FUNCTION_BLOCK ValveBase (* Composite Function Block Type *)
  (* Standard: 61499-2 *)
  (* Version 1.0.1, 10/17/2023, ApplicationLibDevTeam, Schneider Electric, First Version *)
  PACKAGE Main;
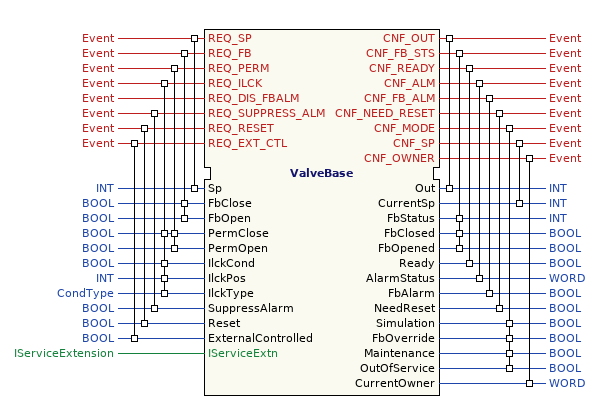
  EVENT_INPUT
    REQ_SP WITH Sp; (* Request to update setpoint *)
    REQ_FB WITH FbClose, FbOpen; (* Request to update feedbacks *)
    REQ_PERM WITH PermClose, PermOpen; (* Request to update permissive conditions *)
    REQ_ILCK WITH PermClose, IlckCond, IlckPos, IlckType; (* Request to update interlock conditions *)
    REQ_DIS_FBALM; (* Request to disable feedback alarm *)
    REQ_SUPPRESS_ALM WITH SuppressAlarm; (* Request to update the alarm suppress status *)
    REQ_RESET WITH Reset; (* Request to reset the device *)
    REQ_EXT_CTL WITH ExternalControlled;
  END_EVENT
  EVENT_OUTPUT
    CNF_OUT WITH Out; (* Execution of confirmation output *)
    CNF_FB_STS WITH FbStatus, FbOpened, FbClosed; (* Execution of confirmed state *)
    CNF_READY WITH Ready; (* Execution of Ready status *)
    CNF_ALM WITH AlarmStatus; (* Execution of confirmation  alarm conditions *)
    CNF_FB_ALM WITH FbAlarm; (* Execution of confirmation  Fb alarm *)
    CNF_NEED_RESET WITH NeedReset; (* Request for Reset *)
    CNF_MODE WITH OutOfService, Simulation, FbOverride, Maintenance; (* Excecution of new operational modes *)
    CNF_SP WITH CurrentSp;
    CNF_OWNER WITH CurrentOwner; (* Execution confirmation of owner *)
  END_EVENT
  VAR_INPUT
    Sp : INT; (* Setpoint of device (1 = Open, 2 = Close) *)
    FbClose : BOOL; (* 1 = Device Close feedback active *)
    FbOpen : BOOL; (* 1 = Device Open feedback active *)
    PermClose : BOOL := TRUE; (* 1 = Device Close permission active *)
    PermOpen : BOOL := TRUE; (* 1 = Device Open permission active *)
    IlckCond : BOOL; (* 1 = Interlock condition active *)
    IlckPos : INT; (* Interlock setpoint state (0 = stop, 1 = Open, 2 = Close, 3 = Interlock inactive) *)
    IlckType : CondType; (* Type of condition interlock, (0 = Normal, 1 = Process interlock/Sequence interlock) *)
    SuppressAlarm : BOOL; (* 1 = Suppress alarm in HMI *)
    Reset : BOOL; (* 1 = Reset device failure *)
    ExternalControlled : BOOL; (* 1 = External control is active *)
  END_VAR
  VAR_OUTPUT
    Out : INT; (* Output to HW ( 1 = Open command, 2 = Close command) depending on NO/NC *)
    CurrentSp : INT; (* Output value considering permissive conditions *)
    FbStatus : INT; (* Confirmed state of the device (0 = Stopped, 1 = Opened, 2 = Closed , 253 = Unknown) *)
    FbClosed : BOOL; (* 1 = Closed *)
    FbOpened : BOOL; (* 1 = Opened *)
    Ready : BOOL; (* 1 = Device is ready to run *)
    AlarmStatus : WORD; (* Bit 2 = Feedback failure status *)
    FbAlarm : BOOL; (* 1 = Feedback failure alarm is active *)
    NeedReset : BOOL; (* 1 = Device need reset to resume the operation *)
    Simulation : BOOL; (* 1 = Simulation mode is active *)
    FbOverride : BOOL; (* 1 = Feedback overide (Sp = FbStatus) *)
    Maintenance : BOOL; (* 1 = Maintenance mode is active *)
    OutOfService : BOOL; (* 1 = Out of service mode is active *)
    CurrentOwner : WORD; (* Current owner data from externlal source and basic owner 16#8 = Program owner, 16#10 = Operator owner, 16#4 = program Local and 16#40 Operator Local *)
  END_VAR
  SOCKETS
    IServiceExtn : IServiceExtension(ServiceState := TRUE); (* Services extension adapter(Seq control, Local panel, Maintenance and Owner) *)
  END_SOCKETS
  (* Alarm Managment *)
  (* Data exchange with sequence *)
  (* Initialization *)
  (* Supervision Interface *)
  (* Owner & Setpoint Management *)
  (* Control *)
  FBS
    plcStart : plcStart(Delay := T#0ms, Prio := 16); {SET_ATTRIBUTE(Configuration.Component.HideUnusedPorts, )}
    spSelection : devInSel(EnBumpless1 := FALSE, EnBumpless2 := TRUE, EnBumpless3 := TRUE, ResetSp := (value:=0,quality:=16#0,timestamp:=LDT#2023-01-20-10:13:38,picosecs:=0), InitialVal := (value:=1,quality:=16#0,timestamp:=LDT#2023-08-11-12:54:59,picosecs:=0)); {SET_ATTRIBUTE(Configuration.Component.HideUnusedPorts, )}
    control : valveLogic;
    feedbackFailure : stateAlarmBasic(AlarmState := TRUE); {SET_ATTRIBUTE(Configuration.Component.HideUnusedPorts, )} {SET_ATTRIBUTE(HMI.AlarmText, $key:SE.App2CommonProcess.AlmLableFbFail)}
    progSpSelection : SELECT_24363B89CFDE21263; {SET_ATTRIBUTE(Configuration.GenericFBType.InterfaceParams, Runtime.Standard#CNT:=2;SELECT:BOOL;IN${CNT$}:INT)}
    IThis : ValveBase_HMI(QI := TRUE);
    basicOwner : ownerControl;
    resetConditions : DS_SELECTX_1579ED5B8ACDFC94C; {SET_ATTRIBUTE(Configuration.GenericFBType.InterfaceParams, Runtime.Standard#CNTX:=3;CNTY:=1;DI${CNTX,_,CNTY$}:BOOL)}
  END_FBS
  EVENT_CONNECTIONS
    control.CNF_FB_ALM TO CNF_FB_ALM;
    control.CNF_FB_STS TO CNF_FB_STS;
    control.CNF_MODE TO CNF_MODE;
    REQ_FB TO control.REQ_FB;
    REQ_DIS_FBALM TO control.REQ_PARA;
    REQ_PERM TO spSelection.REQ_SEL;
    basicOwner.CNF_OWNER TO spSelection.REQ_SEL;
    control.CNF_NEED_RESET TO CNF_NEED_RESET;
    control.CNF_READY TO CNF_READY;
    control.CNF_FB_ALM TO feedbackFailure.REQ;
    control.CNF_ALM TO CNF_ALM;
    control.CNF_OUT TO IServiceExtn.CNF_STATUS;
    control.CNF_FB_STS TO IServiceExtn.CNF_STATUS;
    control.CNF_READY TO IServiceExtn.CNF_READY;
    control.CNF_MODE TO IServiceExtn.CNF_OPMODE;
    REQ_SUPPRESS_ALM TO IServiceExtn.CNF_SUPPRESS_ALM;
    feedbackFailure.INITO TO plcStart.ACK_FIRST;
    plcStart.FIRST_INIT TO IServiceExtn.CNF_SERVICE;
    control.CNF_ILCK TO spSelection.REQ_SEL;
    REQ_SUPPRESS_ALM TO feedbackFailure.REQ_SUPRESS;
    control.CNF_OUT TO CNF_OUT;
    REQ_ILCK TO control.REQ_ILCK;
    spSelection.CNF TO control.REQ_SP;
    IServiceExtn.REQ_OWNER TO basicOwner.REQ_STDOWNER;
    REQ_PERM TO IServiceExtn.CNF_READY;
    control.CNF_DEFAULT_STATE TO spSelection.REQ_SP1;
    REQ_SP TO progSpSelection.REQ;
    IServiceExtn.REQ_CMD TO progSpSelection.REQ;
    progSpSelection.CNF TO spSelection.REQ_SP3;
    control.CNF_ILCK TO IServiceExtn.CNF_READY;
    control.CNF_SP TO CNF_SP;
    control.CNF_ALM TO IServiceExtn.CNF_READY;
    REQ_EXT_CTL TO control.REQ_EXT_CTL;
    basicOwner.CNF_OWNER TO CNF_OWNER;
    REQ_RESET TO resetConditions.REQ3;
    IServiceExtn.REQ_RESET TO resetConditions.REQ2;
    resetConditions.IND TO control.REQ_RESET;
    control.CNF_NEED_RESET TO IServiceExtn.CNF_READY;
    control.CNF_DEFAULT_STATE TO IServiceExtn.CNF_DEFAULT_STATE;
    plcStart.FIRST_INIT TO IThis.34A017503AC1070A;
    IThis.377462E9CE5193B5 TO IThis.F2953B6BB9388F21;
    control.CNF_OUT TO IThis.EC791CA6E67D66B3;
    control.CNF_FB_STS TO IThis.EC791CA6E67D66B3;
    control.CNF_NEED_RESET TO IThis.EC791CA6E67D66B3;
    spSelection.CNF TO IThis.EC791CA6E67D66B3;
    control.CNF_TRANS_FB TO IThis.EC791CA6E67D66B3;
    REQ_SUPPRESS_ALM TO IThis.EC791CA6E67D66B3;
    feedbackFailure.CNF_ALM TO IThis.EC791CA6E67D66B3;
    control.CNF_ILCK TO IThis.EC791CA6E67D66B3;
    REQ_PERM TO IThis.EC791CA6E67D66B3;
    basicOwner.CNF_OWNER TO IThis.EC791CA6E67D66B3;
    control.CNF_SP TO IThis.EC791CA6E67D66B3;
    REQ_EXT_CTL TO IThis.EC791CA6E67D66B3;
    IThis.377462E9CE5193B5 TO feedbackFailure.INIT;
    IThis.377462E9CE5193B5 TO basicOwner.REQ_BASICOWNER;
    IThis.95BEA68906019444 TO feedbackFailure.REQ_PARA;
    IThis.95BEA68906019444 TO control.REQ_DEFAULT_STATE;
    IThis.95BEA68906019444 TO control.REQ_PARA;
    IThis.95BEA68906019444 TO IServiceExtn.CNF_CFG;
    IThis.C6CA4032A5F6989A TO spSelection.REQ_SP2;
    IThis.1A2B085F4B246BF1 TO resetConditions.REQ1;
    IThis.4711DA9A2DFC024 TO control.REQ_PARA;
    IThis.4711DA9A2DFC024 TO spSelection.REQ_SEL;
    IThis.4711DA9A2DFC024 TO basicOwner.REQ_FORCE;
    IThis.AB45C9C76752120B TO basicOwner.REQ_BASICOWNER;
    control.CNF_SP TO IServiceExtn.CNF_STATUS;
  END_CONNECTIONS
  DATA_CONNECTIONS
    control.FbAlarm TO FbAlarm;
    control.Mode TO IServiceExtn.OpMode;
    SuppressAlarm TO feedbackFailure.Suppress;
    control.FbAlarm TO feedbackFailure.Input;
    IlckType TO control.IlckType;
    FbClose TO control.FbClose;
    FbOpen TO control.FbOpen;
    control.FbClosed TO FbClosed;
    control.FbOpened TO FbOpened;
    control.FbStatus TO FbStatus;
    control.NeedReset TO NeedReset;
    control.Ready TO Ready;
    control.Alarm TO AlarmStatus;
    control.CurrentSp TO CurrentSp;
    control.FbStatus TO IServiceExtn.Status;
    control.CurrentSp TO IServiceExtn.CurrentSp;
    control.CurrentOut TO IServiceExtn.CurrentOp;
    control.NeedReset TO IServiceExtn.NeedReset;
    control.Ready TO IServiceExtn.Ready;
    SuppressAlarm TO IServiceExtn.SuppressAlarm;
    control.CondPos TO spSelection.IlckSp;
    control.Interlocked TO spSelection.Ilck;
    control.Out TO Out;
    IlckPos TO control.IlckPos;
    PermClose TO spSelection.PermActive2;
    IlckCond TO control.IlckCond;
    IServiceExtn.StdOwner TO basicOwner.StdOwner;
    basicOwner.OperatorOwner TO spSelection.Sel2;
    basicOwner.ProgramOwner TO spSelection.Sel3;
    control.Alarm TO IServiceExtn.Alarm;
    control.Interlocked TO IServiceExtn.Interlocked;
    PermOpen TO IServiceExtn.PermActive1;
    PermClose TO IServiceExtn.PermActive2;
    PermClose TO spSelection.PermPassive;
    control.DefaultState TO spSelection.Val1;
    basicOwner.StdOwnerConnected TO progSpSelection.SELECT;
    Sp TO progSpSelection.IN1;
    IServiceExtn.Sp TO progSpSelection.IN2;
    progSpSelection.OUT TO spSelection.Val3;
    spSelection.PermVal TO control.Sp;
    PermClose TO IServiceExtn.PermPassive;
    ExternalControlled TO control.ExternalControlled;
    basicOwner.Owner TO CurrentOwner;
    Reset TO resetConditions.DI3_1;
    IServiceExtn.Reset TO resetConditions.DI2_1;
    resetConditions.OUT1 TO control.Reset;
    control.DefaultState TO IServiceExtn.DefaultState;
    PermOpen TO spSelection.PermActive1;
    control.FbStatus TO IThis.F2AD3CD6DCE76874;
    control.TransFbStatus TO IThis.18339E8B84CEF55;
    control.CurrentOut TO IThis.D2C35BC47DF71FCC;
    control.CurrentSp TO IThis.C6876D790F3A950E;
    control.NeedReset TO IThis.9CD6749867E91606;
    basicOwner.Owner TO IThis.66F5D611520B8E21;
    feedbackFailure.AlarmStatus TO IThis.E324EF7311434CB7;
    control.Interlocked TO IThis.CAD2FBF5C8122C72;
    control.CondPos TO IThis.F97E56AEBDD59492;
    PermClose TO IThis.7DE7E04BA65FF582;
    PermOpen TO IThis.F1D46CDCC1D5A6C6;
    basicOwner.StdOwnerConnected TO IThis.9BBC553B7236462E;
    ExternalControlled TO IThis.6C32AB699640FC5A;
    IThis.D82AC87A2FA22E86 TO basicOwner.BasicOwner;
    IThis.861B8773AF2757FC TO control.MonTime;
    IThis.5568E3E91B9AAED8 TO control.TripTime;
    IThis.3DA6D0F9276D43A4 TO control.ConfResetReq;
    IThis.4D34C1A4533BA5DF TO resetConditions.DI1_1;
    IThis.869E02415F6A841 TO spSelection.Val2;
    IThis.CF1EA84FDDBF53A1 TO control.Simulation;
    IThis.CF1EA84FDDBF53A1 TO Simulation;
    IThis.AD38F01F8F0043E7 TO control.FbOverride;
    IThis.AD38F01F8F0043E7 TO FbOverride;
    IThis.C8DEEF765E4F14C0 TO control.Maintenance;
    IThis.C8DEEF765E4F14C0 TO Maintenance;
    IThis.C8DEEF765E4F14C0 TO basicOwner.ForceOperator;
    IThis.C4714A0B76119976 TO control.OutOfService;
    IThis.C4714A0B76119976 TO OutOfService;
    IThis.C4714A0B76119976 TO spSelection.Sel1;
    IThis.B394B8C6484B76DE TO feedbackFailure.ScanTime;
    IThis.E4ACFA19543211CB TO feedbackFailure.AckType;
    IThis.52A3AF601F61E85C TO spSelection.EnTrackSp;
    IThis.52A3AF601F61E85C TO IServiceExtn.EnTrackSp;
    IThis.6A4CE6BC8D982056 TO control.SelDefaultState;
    IThis.6A4CE6BC8D982056 TO control.ValveCmdType;
    IThis.6A4CE6BC8D982056 TO spSelection.EnInitialVal;
    IThis.7801A8D91AA682F9 TO control.FbMode;
  END_CONNECTIONS
END_FUNCTION_BLOCK
